TYPE InputBase_8311D824 : 
STRUCT
END_STRUCT
END_TYPE

(* stored: Version 1.1.0.1, ProductVersion 3.1.4024.9
   DUT InputBase_8311D824: Id {d437bbc9-c12a-0ffe-2f34-2f36901f67f9} *)
